Staubli VAL3: cartStatus.pgx

public program cartStatus(num x_nCartConnFlag, num x_nLastMsgAge)
begin

  // Do nothing
  // See start() program for more details

end
